FUNCTION_BLOCK SS4_ifb_Raiser_n_Flipper (* Basic FB with empty ECC *)
  (* Standard: 61499-2 *)
  (* Version 1.0, 2021-08-23, AK121668 *)
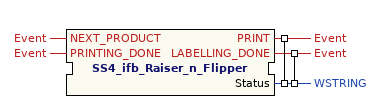
  EVENT_INPUT
    NEXT_PRODUCT;
    PRINTING_DONE;
  END_EVENT
  EVENT_OUTPUT
    PRINT WITH Status;
    LABELLING_DONE WITH Status;
  END_EVENT
  VAR_OUTPUT
    Status : WSTRING;
  END_VAR
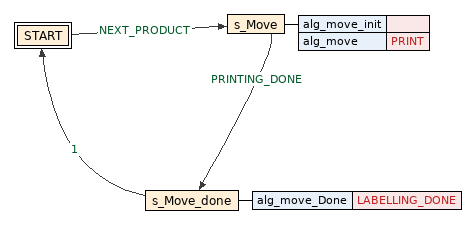
  EC_STATES
    START; (* Initial State *)
    s_Move : alg_move_init, alg_move -> PRINT;
    s_Move_done : alg_move_Done -> LABELLING_DONE;
  END_STATES
  EC_TRANSITIONS
    s_Move_done TO START := 1;
    START TO s_Move := NEXT_PRODUCT;
    s_Move TO s_Move_done := PRINTING_DONE;
  END_TRANSITIONS
  ALGORITHM alg_move_init IN ST:

  END_ALGORITHM
  ALGORITHM alg_move IN ST:
Status := "Lasering Start";
  END_ALGORITHM
  ALGORITHM alg_move_Done IN ST:
Status := "Lasering DONE";
  END_ALGORITHM
END_FUNCTION_BLOCK
